(* IEC 61131-3 sources: SRCI/RobotLibrary/Library/Functions/Check, 7 files *)

(* ---- IsDefaultDynamicsEqual.st ---- *)
FUNCTION IsDefaultDynamicsEqual : BOOL
// -------------------------------------------------------------------------
//  SRCI Robot Library
// -------------------------------------------------------------------------
//
//  Object:      IsDefaultDynamicsEqual
//  Author:      Thorsten Brach
//  Date:        2025-04-23
//
//  Description:
//
//
//  Copyright:
//    (C) 2025 Thorsten Brach. All rights reserved
//             Licensed under the LGPL-3.0 license.
//
//  Disclaimer:
//    This project is provided without any guarantee and can be used for
//    private and commercial purposes. Any use is at the user’s
//    own risk and responsibility.
//
// -------------------------------------------------------------------------
VAR_INPUT
  /// DefaultDynamics 1 to compare
  Data1           : DefaultDynamics;
  /// DefaultDynamics 2 to compare
  Data2           : DefaultDynamics;
  /// Flag to ignore the timestamp during the comparison
  IgnoreTimestamp : BOOL;
END_VAR

  IF (IgnoreTimestamp)
  THEN
    Data1.Timestamp := Data2.Timestamp;
  END_IF

  IsDefaultDynamicsEqual := ( SysDepMemCmp( pData1 := ADR(Data1), pData2 :=  ADR(Data2), DataLen := SIZEOF(Data1)) = RobotLibraryConstants.OK );

END_FUNCTION

(* ---- IsFrameDataEqual.st ---- *)
FUNCTION IsFrameDataEqual : BOOL
// -------------------------------------------------------------------------
//  SRCI Robot Library
// -------------------------------------------------------------------------
//
//  Object:      IsFrameDataEqual
//  Author:      Thorsten Brach
//  Date:        2025-04-23
//
//  Description:
//
//
//  Copyright:
//    (C) 2025 Thorsten Brach. All rights reserved
//             Licensed under the LGPL-3.0 license.
//
//  Disclaimer:
//    This project is provided without any guarantee and can be used for
//    private and commercial purposes. Any use is at the user’s
//    own risk and responsibility.
//
// -------------------------------------------------------------------------
VAR_INPUT
  /// FrameData 1 to compare
  Data1           : FrameData;
  /// FrameData 2 to compare
  Data2           : FrameData;
  /// Flag to ignore the timestamp during the comparison
  IgnoreTimestamp : BOOL;
END_VAR

  IF (IgnoreTimestamp)
  THEN
    Data1.Timestamp := Data2.Timestamp;
  END_IF

  IsFrameDataEqual := ( SysDepMemCmp( pData1 := ADR(Data1), pData2 :=  ADR(Data2), DataLen := SIZEOF(Data1)) = RobotLibraryConstants.OK );

END_FUNCTION

(* ---- IsLoadDataEqual.st ---- *)
FUNCTION IsLoadDataEqual : BOOL
// -------------------------------------------------------------------------
//  SRCI Robot Library
// -------------------------------------------------------------------------
//
//  Object:      IsLoadDataEqual
//  Author:      Thorsten Brach
//  Date:        2025-04-23
//
//  Description:
//
//
//  Copyright:
//    (C) 2025 Thorsten Brach. All rights reserved
//             Licensed under the LGPL-3.0 license.
//
//  Disclaimer:
//    This project is provided without any guarantee and can be used for
//    private and commercial purposes. Any use is at the user’s
//    own risk and responsibility.
//
// -------------------------------------------------------------------------
VAR_INPUT
  /// LoadData 1 to compare
  Data1           : LoadData;
  /// LoadData 2 to compare
  Data2           : LoadData;
  /// Flag to ignore the timestamp during the comparison
  IgnoreTimestamp : BOOL;
END_VAR

  IF (IgnoreTimestamp)
  THEN
    Data1.Timestamp := Data2.Timestamp;
  END_IF

  IsLoadDataEqual := ( SysDepMemCmp( pData1 := ADR(Data1), pData2 :=  ADR(Data2), DataLen := SIZEOF(Data1)) = RobotLibraryConstants.OK );

END_FUNCTION

(* ---- IsReferenceDynamicsEqual.st ---- *)
FUNCTION IsReferenceDynamicsEqual : BOOL
// -------------------------------------------------------------------------
//  SRCI Robot Library
// -------------------------------------------------------------------------
//
//  Object:      IsReferenceDynamicsEqual
//  Author:      Thorsten Brach
//  Date:        2025-04-23
//
//  Description:
//
//
//  Copyright:
//    (C) 2025 Thorsten Brach. All rights reserved
//             Licensed under the LGPL-3.0 license.
//
//  Disclaimer:
//    This project is provided without any guarantee and can be used for
//    private and commercial purposes. Any use is at the user’s
//    own risk and responsibility.
//
// -------------------------------------------------------------------------
VAR_INPUT
  /// ReferenceDynamics 1 to compare
  Data1           : ReferenceDynamics;
  /// ReferenceDynamics 2 to compare
  Data2           : ReferenceDynamics;
  /// Flag to ignore the timestamp during the comparison
  IgnoreTimestamp : BOOL;
END_VAR

  IF (IgnoreTimestamp)
  THEN
    Data1.Timestamp := Data2.Timestamp;
  END_IF

  IsReferenceDynamicsEqual := ( SysDepMemCmp( pData1 := ADR(Data1), pData2 :=  ADR(Data2), DataLen := SIZEOF(Data1)) = RobotLibraryConstants.OK );

END_FUNCTION

(* ---- IsSwLimitsEqual.st ---- *)
FUNCTION IsSwLimitsEqual : BOOL
// -------------------------------------------------------------------------
//  SRCI Robot Library
// -------------------------------------------------------------------------
//
//  Object:      IsSwLimitsEqual
//  Author:      Thorsten Brach
//  Date:        2025-04-23
//
//  Description:
//
//
//  Copyright:
//    (C) 2025 Thorsten Brach. All rights reserved
//             Licensed under the LGPL-3.0 license.
//
//  Disclaimer:
//    This project is provided without any guarantee and can be used for
//    private and commercial purposes. Any use is at the user’s
//    own risk and responsibility.
//
// -------------------------------------------------------------------------
VAR_INPUT
  /// SW Limit 1 to compare
  Data1           : SWLimits;
  /// SW LIMIT 2 to compare
  Data2           : SWLimits;
  /// Flag to ignore the timestamp during the comparison
  IgnoreTimestamp : BOOL;
END_VAR

  IF (IgnoreTimestamp)
  THEN
    Data1.Timestamp := Data2.Timestamp;
  END_IF

  IsSwLimitsEqual := ( SysDepMemCmp( pData1 := ADR(Data1), pData2 :=  ADR(Data2), DataLen := SIZEOF(Data1)) = RobotLibraryConstants.OK );

END_FUNCTION

(* ---- IsToolDataEqual.st ---- *)
FUNCTION IsToolDataEqual : BOOL
// -------------------------------------------------------------------------
//  SRCI Robot Library
// -------------------------------------------------------------------------
//
//  Object:      IsToolDataEqual
//  Author:      Thorsten Brach
//  Date:        2025-04-23
//
//  Description:
//
//
//  Copyright:
//    (C) 2025 Thorsten Brach. All rights reserved
//             Licensed under the LGPL-3.0 license.
//
//  Disclaimer:
//    This project is provided without any guarantee and can be used for
//    private and commercial purposes. Any use is at the user’s
//    own risk and responsibility.
//
// -------------------------------------------------------------------------
VAR_INPUT
  /// ToolData 1 to compare
  Data1           : ToolData;
  /// ToolData 2 to compare
  Data2           : ToolData;
  /// Flag to ignore the timestamp during the comparison
  IgnoreTimestamp : BOOL;
END_VAR

  IF (IgnoreTimestamp)
  THEN
    Data1.Timestamp := Data2.Timestamp;
  END_IF

  IsToolDataEqual := ( SysDepMemCmp( pData1 := ADR(Data1), pData2 :=  ADR(Data2), DataLen := SIZEOF(Data1)) = RobotLibraryConstants.OK );

END_FUNCTION

(* ---- IsWorkAreaEqual.st ---- *)
FUNCTION IsWorkAreaEqual : BOOL
// -------------------------------------------------------------------------
//  SRCI Robot Library
// -------------------------------------------------------------------------
//
//  Object:      IsWorkAreaEqual
//  Author:      Thorsten Brach
//  Date:        2025-04-23
//
//  Description:
//
//
//  Copyright:
//    (C) 2025 Thorsten Brach. All rights reserved
//             Licensed under the LGPL-3.0 license.
//
//  Disclaimer:
//    This project is provided without any guarantee and can be used for
//    private and commercial purposes. Any use is at the user’s
//    own risk and responsibility.
//
// -------------------------------------------------------------------------
VAR_INPUT
  /// WorkArea 1 to compare
  Data1           : RobotWorkAreaData;
  /// WorkArea 2 to compare
  Data2           : RobotWorkAreaData;
  /// Flag to ignore the timestamp during the comparison
  IgnoreTimestamp : BOOL;
END_VAR

  IF (IgnoreTimestamp)
  THEN
    Data1.Timestamp := Data2.Timestamp;
  END_IF

  IsWorkAreaEqual := ( SysDepMemCmp( pData1 := ADR(Data1), pData2 :=  ADR(Data2), DataLen := SIZEOF(Data1)) = RobotLibraryConstants.OK );

END_FUNCTION
